FUNCTION_BLOCK fbPistonMoveTask EXTENDS TcoCore.TcoTask
VAR_INPUT
	PositionSensor : BOOL;
END_VAR
VAR_IN_OUT
	MoveToPositionSignal : BOOL;
	InverseSignal : BOOL;	
END_VAR

IF(THIS^.Execute())THEN
	THIS^.Messenger.Debug('Executing piston movement');
	InverseSignal := FALSE;
	MoveToPositionSignal := TRUE;
	THIS^.DoneWhen(PositionSensor);
END_IF

END_FUNCTION_BLOCK

(* stored: Version 1.1.0.1, ProductVersion 3.1.4024.6
   POU fbPistonMoveTask: Id {b9f74900-963d-0b1a-2103-6fbbac7ef37b}, SpecialFunc None *)
